// TIA Portal V20 export
DATA_BLOCK "DI1"   // DB279
// stored: MemoryReserve 100
   VAR
      "MOTOR POWER TRIPPED E202CB" : Bool;
      "REELCUT CONVEYOR RING BLOW POWER TRIPPED" : Bool;
      "STACKING-1 CONVEYOR RING BLOW POWER TRIPPED E214CB" : Bool;
      "STACKING-2 CONVEYOR RING BLOW POWER TRIPPED E220CB" : Bool;
      SPARE1 : Bool;
      "E6404PWS CONTROLLER POWER SMPS AC POWER TRIPPED E320CB" : Bool;
      "E6704PWS CONTROLLER POWER SMPS AC POWER TRIPPED E326CB" : Bool;
      "E6804PWS SAFETY POWER SMPS AC POWER TRIPPED E332CB" : Bool;
      SPARE2 : Bool;
      "POWER METER POWER TRIPPED E720CB" : Bool;
      "POWER METER CONTROL POWER TRIPPED E726CB" : Bool;
      SPARE3 : Bool;
      "PROCESSOR POWER ON TRIPPED E4116CB" : Bool;
      "PROGRAMMING POWER OUTLET TRIPPED E4156CB" : Bool;
      SPARE4 : Bool;
      "PANEL LED POWER TRIPPED E4304CB" : Bool;
      SPARE5 : Bool;
      "PLC POWER SMPS DC OK E4404PWS" : Bool;
      "CONTROL LEVEL HUB POWER TRIPPED E4420CB" : Bool;
      "MAIN HMI POWER TRIPPED E4426CB" : Bool;
      "PORTABLE HMI POWER TRIPPED E4432CB" : Bool;
      "PORTABLE HMI POWER TRIPPED E4456CB" : Bool;
      SPARE6 : Bool;
      SPARE7 : Bool;
      "120VAC CONTROL POWER TR PRIMARY TRIPPED E5100CB" : Bool;
      "120VAC CONTROL POWER TR SECONDARY TRIPPED E5110CB" : Bool;
      "CONTROL POWER ON TRIPPED E5116CB" : Bool;
      "VISION MONITOR POWER STRIP OUTLET POWER TRIPPED E5160CB" : Bool;
      "MCU & RFD HANDY POWER STRIP OUTLET POWER TRIPPED E5166CB" : Bool;
      "VISION LIGHT CONTROLLER POWER STRIP OUTLET POWER TRIPPED E5172CB" : Bool;
      SPARE8 : Bool;
      "FFU POWER-1 POWER TRIPPED E3222CB" : Bool;
   END_VAR
BEGIN
END_DATA_BLOCK
